FUNCTION_BLOCK FB_StateMachine
VAR_INPUT
    EnableIn : BOOL;
    cfgAutoRun : BOOL;
    inpBlockedCondition : DINT;
    inpStarvedCondition : DINT;
    inpSubmoduleFaulted : BOOL;
END_VAR

VAR_OUTPUT
    EnableOut : BOOL;
    Status : ST_SM_Status;
END_VAR

VAR CONSTANT
    HOMING_MIN   : DINT := 1000; HOMING_MAX   : DINT := 1999;
    RUNNING_MIN  : DINT := 3000; RUNNING_MAX  : DINT := 3999;
    STOPPING_MIN : DINT := 2000; STOPPING_MAX : DINT := 2999;
    ABORTING_MIN : DINT := 5000; ABORTING_MAX : DINT := 5999;
    PAUSING_MIN  : DINT := 4000; PAUSING_MAX  : DINT := 4999;
    PROCEEDING_MIN : DINT := 6000; PROCEEDING_MAX : DINT := 6999;
END_VAR

VAR
    // Internal command request flags (set by methods, consumed by body)
    _abortRequested : BOOL;
    _completeStateRequested : BOOL;
    _homeRequested : BOOL;
    _pauseRequested : BOOL;
    _proceedRequested : BOOL;
    _startRequested : BOOL;
    _stopRequested : BOOL;
    _retryActive : BOOL;
    RetryComplete : BOOL;
    
    // Timer
    StepTimer : TON;
    
    // Edge detection
    R_TRIG_1 : R_TRIG;
    R_TRIG_5 : R_TRIG;
    
    // Internal state tracking
    _previousState : E_SM_State;
    PreviousStep : DINT;
    TimerReset : BOOL;
    LsOdd : DINT;
    _returnState : E_SM_State;
    ReturnNextStep : DINT;
    
    // Permission handlers
    permAuto : FB_Permissives;
    permHome : FB_Permissives;
    permProceed : FB_Permissives;
    permStart : FB_Permissives;
    
    // Running interlock (latching - auto-aborts from any active state)
    intlkRunning : FB_Interlock;
    
    // Temp variables
    permIndex : UDINT;
    stepIsZero : BOOL;
    seqDone : BOOL;
    
    // Source control
    bSourceLockedToProg : BOOL;
    
    // Step ownership (internal)
    _nextStep : DINT;
END_VAR


//-----------------------------------------------------------------------------
// Main Implementation
//-----------------------------------------------------------------------------
EnableOut := EnableIn;

// Only execute if enabled
IF EnableIn THEN
    //-------------------------------------------------------------------------
    // Process permissions for different states
    //-------------------------------------------------------------------------
    permHome();
    permStart();
    permProceed();
    permAuto();
    
    intlkRunning();
    
    // Auto-abort if any running interlock trips (e-stop, safety gate, etc.)
    IF NOT intlkRunning.sts.bOK AND
       NOT (Status.State = E_SM_State.STOPPED OR Status.State = E_SM_State.ABORTING) THEN
        _abortRequested := TRUE;
    END_IF;
    
    //-------------------------------------------------------------------------
    // Ready state calculations
    //-------------------------------------------------------------------------
    Status.ReadyToHome := (Status.State = E_SM_State.STOPPED) AND
                          permHome.sts.bOK AND
                          permAuto.sts.bOK;

    Status.ReadyToStart := (Status.State = E_SM_State.READY) AND
                          permStart.sts.bOK AND
                          permAuto.sts.bOK AND
                          NOT Status.AutoStartRequest;

    Status.ReadyToProceed := (Status.State = E_SM_State.PAUSED) AND
                            permProceed.sts.bOK AND
                            permAuto.sts.bOK;

    //-------------------------------------------------------------------------
    // Auto-start request logic
    // AutoCycle fires when we just finished a RUNNING cycle (READY with LastState=RUNNING)
    //-------------------------------------------------------------------------
    Status.AutoStartRequest := _startRequested AND NOT permStart.sts.bOK;
    Status.AutoCycleRequest := cfgAutoRun AND (Status.State = E_SM_State.READY) AND
                              (Status.LastState = E_SM_State.RUNNING) AND NOT permStart.sts.bOK;

    //-------------------------------------------------------------------------
    // Remember last state before change
    //-------------------------------------------------------------------------
    _previousState := Status.State;

    //-------------------------------------------------------------------------
    // Auto-run handling (internal - not from external command)
    //-------------------------------------------------------------------------
    IF cfgAutoRun AND permAuto.sts.bOK AND permStart.sts.bOK AND
       (Status.State = E_SM_State.READY) AND (Status.LastState = E_SM_State.RUNNING) THEN
        _startRequested := TRUE;
    END_IF;
    
    //-------------------------------------------------------------------------
    // Sequence completion inference
    //-------------------------------------------------------------------------
    seqDone := _IsStepInStateRange(
        state := Status.State,
        nStep := Status.Step.Current
    ) AND (_nextStep = 0);

    R_TRIG_5(CLK := seqDone);
    IF R_TRIG_5.Q THEN
        _completeStateRequested := TRUE;
    END_IF;

    //-------------------------------------------------------------------------
    // State Transitions
    //-------------------------------------------------------------------------

    // Homing complete → Ready
    IF _completeStateRequested AND (Status.State = E_SM_State.HOMING) THEN
        _nextStep := 0;
        Status.State := E_SM_State.READY;
        _completeStateRequested := FALSE;
    END_IF;

    // Running complete → Ready (LastState will be RUNNING so AutoCycle can detect a just-finished cycle)
    IF _completeStateRequested AND (Status.State = E_SM_State.RUNNING) THEN
        _nextStep := 0;
        Status.State := E_SM_State.READY;
        _completeStateRequested := FALSE;
    END_IF;

    // Running + Stop → Stopping
    IF _stopRequested AND (Status.State = E_SM_State.RUNNING) THEN
        Status.State := E_SM_State.STOPPING;
    END_IF;

    // Stopping complete → Stopped
    IF _completeStateRequested AND (Status.State = E_SM_State.STOPPING) THEN
        _nextStep := 0;
        Status.State := E_SM_State.STOPPED;
        _completeStateRequested := FALSE;
    END_IF;

    // Aborting complete → Stopped (Status.Faulted remains indicated via LastState = ABORTING)
    IF _completeStateRequested AND (Status.State = E_SM_State.ABORTING) THEN
        _nextStep := 0;
        Status.State := E_SM_State.STOPPED;
        _completeStateRequested := FALSE;
    END_IF;

    // Running + Pause → Pausing (save context for Proceed)
    IF _pauseRequested AND (Status.State = E_SM_State.RUNNING) THEN
        _returnState := Status.State;
        ReturnNextStep := Status.Step.Current;  // resume re-enters same step
        Status.State := E_SM_State.PAUSING;
        _nextStep := 0;
    END_IF;

    // Pausing complete → Paused
    IF _completeStateRequested AND (Status.State = E_SM_State.PAUSING) THEN
        _nextStep := 0;
        Status.State := E_SM_State.PAUSED;
        _completeStateRequested := FALSE;
    END_IF;

    // Proceeding complete → return to state before pause, re-enter the paused step
    IF _completeStateRequested AND (Status.State = E_SM_State.PROCEEDING) THEN
        _nextStep := ReturnNextStep;
        Status.State := _returnState;
        _completeStateRequested := FALSE;
    END_IF;

    // Ready + Start → Running
    IF (_startRequested OR
        (Status.AutoStartRequest AND permStart.sts.bOK AND permAuto.sts.bOK)) AND
        (Status.State = E_SM_State.READY) THEN
        _nextStep := 0;
        Status.State := E_SM_State.RUNNING;
        _startRequested := FALSE;
    END_IF;

    // Ready + Stop → Stopped (no sequence needed, machine is already quiescent)
    IF _stopRequested AND (Status.State = E_SM_State.READY) THEN
        _nextStep := 0;
        Status.State := E_SM_State.STOPPED;
    END_IF;

    // Stopped + Home → Homing
    IF _homeRequested AND (Status.State = E_SM_State.STOPPED) THEN
        _nextStep := 0;
        Status.State := E_SM_State.HOMING;
    END_IF;

    // Paused + Proceed → Proceeding
    IF _proceedRequested AND (Status.State = E_SM_State.PAUSED) THEN
        _nextStep := 0;
        Status.State := E_SM_State.PROCEEDING;
    END_IF;

    // Abort from any state except Stopped / Aborting
    IF _abortRequested AND NOT (Status.State = E_SM_State.STOPPED OR Status.State = E_SM_State.ABORTING) THEN
        _nextStep := 0;
        Status.State := E_SM_State.ABORTING;
    END_IF;
    
    //-------------------------------------------------------------------------
    // Track state changes
    //-------------------------------------------------------------------------
    IF Status.State <> _previousState THEN
        Status.LastState := _previousState;
    END_IF;
    
    //-------------------------------------------------------------------------
    // Derived status flags
    //-------------------------------------------------------------------------
    Status.WaitingState := (Status.State = E_SM_State.STOPPED) OR (Status.State = E_SM_State.READY) OR
                           (Status.State = E_SM_State.PAUSED);
    Status.ActiveState  := (Status.State = E_SM_State.HOMING) OR (Status.State = E_SM_State.RUNNING) OR
                           (Status.State = E_SM_State.STOPPING) OR (Status.State = E_SM_State.PAUSING) OR
                           (Status.State = E_SM_State.PROCEEDING) OR (Status.State = E_SM_State.ABORTING);

    //-------------------------------------------------------------------------
    // Step and timer management
    //-------------------------------------------------------------------------
    
    // Reset timer and clear step name when transitioning to step 0
    stepIsZero := (Status.Step.Current = 0);
    R_TRIG_1(CLK := stepIsZero);
    IF R_TRIG_1.Q THEN
        Status.Step.Name := '';
        _ClearStepPermissives();
        TimerReset := TRUE;
        StepTimer(IN := FALSE, PT := T#99H);
        Status.Step.TimerSeconds := 0.0;
    END_IF;
    
    // Auto-initialize first step when entering an active state
    IF Status.Step.Current = 0 AND Status.ActiveState THEN
        _nextStep := _GetFirstStepForState(state := Status.State);
    END_IF;
    
    // Detect step change and update
    IF Status.Step.Current <> _nextStep THEN
        PreviousStep := Status.Step.Current;
        Status.Step.Current := _nextStep;
        TimerReset := TRUE;
        StepTimer(IN := FALSE, PT := T#99H);
        Status.Step.TimerSeconds := 0.0;
    END_IF;
    
    Status.Step.Next := _nextStep;
    
    // Step timer logic
    IF NOT (Status.State = E_SM_State.PAUSED) OR ((Status.State = E_SM_State.PAUSED) AND _completeStateRequested) THEN
        IF TimerReset THEN
            StepTimer(IN := FALSE, PT := T#99H);
            Status.Step.TimerSeconds := 0.0;
            TimerReset := FALSE;
        ELSE
            StepTimer(IN := TRUE, PT := T#99H);
            Status.Step.TimerSeconds := UDINT_TO_REAL(TIME_TO_UDINT(StepTimer.ET)) / 1000.0;
        END_IF;
    ELSE
        StepTimer(IN := FALSE, PT := T#99H);
    END_IF;
    
    //-------------------------------------------------------------------------
    // Fault detection
    //-------------------------------------------------------------------------
    LsOdd := Status.Step.Current MOD 2;
    Status.Faulted := LsOdd <> 0;
    Status.SubmoduleFaulted := inpSubmoduleFaulted;
    
    //-------------------------------------------------------------------------
    // Retry logic
    //-------------------------------------------------------------------------
    IF RetryComplete THEN
        _retryActive := FALSE;
        RetryComplete := FALSE;
    END_IF;
    
    IF _retryActive THEN
        RetryComplete := TRUE;
    END_IF;
    
    IF _retryActive AND Status.Faulted THEN
        // Roll back to previous (even, non-faulted) step to re-enter it
        _nextStep := Status.Step.Current - 1;
    END_IF;
    
    //-------------------------------------------------------------------------
    // OEE condition codes (Blocked / Starved)
    //-------------------------------------------------------------------------
    IF inpBlockedCondition = 0 THEN
        Status.BlockedCondition := 0;
    END_IF;
    
    IF inpBlockedCondition <> 0 AND
       (Status.State = E_SM_State.RUNNING OR Status.State = E_SM_State.STOPPING OR
        Status.State = E_SM_State.READY) THEN
        Status.BlockedCondition := inpBlockedCondition;
        inpBlockedCondition := 0;
    END_IF;
    
    IF inpStarvedCondition = 0 THEN
        Status.StarvedCondition := 0;
    END_IF;
    
    IF inpStarvedCondition <> 0 AND
       (Status.State = E_SM_State.RUNNING OR Status.State = E_SM_State.STOPPING OR
        Status.State = E_SM_State.READY) THEN
        Status.StarvedCondition := inpStarvedCondition;
        inpStarvedCondition := 0;
    END_IF;
    
ELSE
    // Reset command requests when disabled
    _startRequested := FALSE;
    _stopRequested := FALSE;
    _homeRequested := FALSE;
    _abortRequested := FALSE;
    _pauseRequested := FALSE;
    _proceedRequested := FALSE;
    _completeStateRequested := FALSE;
    Status.Step.Name := '';
        _ClearStepPermissives();
END_IF;

METHOD PRIVATE _ClearStepPermissives
Status.Step.PermCfg.nBypassable := 0;
Status.Step.PermStatus.bOK := FALSE;
Status.Step.PermStatus.nPermissives := 0;
Status.Step.PermStatus.nBypassMask := 0;
Status.Step.PermStatus.nFirstFailureBitIndex := 999;

FOR permIndex := 0 TO 63 DO
        Status.Step.PermCfg.aNames[permIndex] := '';
        Status.Step.PermStatus.aFaceplates[permIndex].name := '';
        Status.Step.PermStatus.aFaceplates[permIndex].stsOK := FALSE;
        Status.Step.PermStatus.aFaceplates[permIndex].stsMapped := FALSE;
        Status.Step.PermStatus.aFaceplates[permIndex].stsBypassed := FALSE;
        Status.Step.PermStatus.aFaceplates[permIndex].cfgBypassable := FALSE;
END_FOR;
END_METHOD

METHOD PRIVATE _GetFirstStepForState : DINT
VAR_INPUT
        state : E_SM_State;
END_VAR
CASE state OF
        E_SM_State.HOMING:     _GetFirstStepForState := HOMING_MIN;
        E_SM_State.RUNNING:    _GetFirstStepForState := RUNNING_MIN;
        E_SM_State.STOPPING:   _GetFirstStepForState := STOPPING_MIN;
        E_SM_State.ABORTING:   _GetFirstStepForState := ABORTING_MIN;
        E_SM_State.PAUSING:    _GetFirstStepForState := PAUSING_MIN;
        E_SM_State.PROCEEDING: _GetFirstStepForState := PROCEEDING_MIN;
ELSE
        _GetFirstStepForState := 0;
END_CASE;
END_METHOD

METHOD PRIVATE _GetLastStepForState : DINT
VAR_INPUT
        state : E_SM_State;
END_VAR
CASE state OF
        E_SM_State.HOMING:     _GetLastStepForState := HOMING_MAX;
        E_SM_State.RUNNING:    _GetLastStepForState := RUNNING_MAX;
        E_SM_State.STOPPING:   _GetLastStepForState := STOPPING_MAX;
        E_SM_State.ABORTING:   _GetLastStepForState := ABORTING_MAX;
        E_SM_State.PAUSING:    _GetLastStepForState := PAUSING_MAX;
        E_SM_State.PROCEEDING: _GetLastStepForState := PROCEEDING_MAX;
ELSE
        _GetLastStepForState := 0;
END_CASE;
END_METHOD

METHOD PRIVATE _IsStepInStateRange : BOOL
VAR_INPUT
        state : E_SM_State;
        nStep : DINT;
END_VAR
_IsStepInStateRange := (nStep >= _GetFirstStepForState(state := state)) AND
                                             (nStep <= _GetLastStepForState(state := state));
END_METHOD

{attribute 'TcRpcEnable' := '1'}
METHOD Abort : E_RpcMethodResponse
VAR_INPUT
    eRequester : E_Requester := E_Requester.PROG;
END_VAR
// Safety command - skip source check, skip fault check
IF Status.State = E_SM_State.STOPPED OR Status.State = E_SM_State.ABORTING THEN
    Abort := E_RpcMethodResponse.REJECTED_WRONG_STATE;
    RETURN;
END_IF;

// Execute - clear other requests, set abort
_startRequested := FALSE;
_stopRequested := FALSE;
_homeRequested := FALSE;
_pauseRequested := FALSE;
_proceedRequested := FALSE;
_completeStateRequested := FALSE;
_abortRequested := TRUE;
Abort := E_RpcMethodResponse.ACCEPTED;
END_METHOD

{attribute 'TcRpcEnable' := '1'}
METHOD Home : E_RpcMethodResponse
VAR_INPUT
    eRequester : E_Requester := E_Requester.PROG;
END_VAR
// Common validation
Home := F_ValidateRequester(eRequester, bSourceLockedToProg, Status.Faulted, FALSE, FALSE);
IF Home <> E_RpcMethodResponse.ACCEPTED THEN RETURN; END_IF;

// State check
IF NOT (Status.State = E_SM_State.STOPPED) THEN
    Home := E_RpcMethodResponse.REJECTED_WRONG_STATE;
    RETURN;
END_IF;

// Permission check (Home-specific)
IF NOT permHome.sts.bOK THEN
    Home := E_RpcMethodResponse.REJECTED_PERMISSIVE_NOT_MET;
    RETURN;
END_IF;

// Permission check (global auto permissives)
IF NOT permAuto.sts.bOK THEN
    Home := E_RpcMethodResponse.REJECTED_PERMISSIVE_NOT_MET;
    RETURN;
END_IF;

// Execute
_abortRequested := FALSE;
_pauseRequested := FALSE;
_proceedRequested := FALSE;
_startRequested := FALSE;
_stopRequested := FALSE;
_completeStateRequested := FALSE;
_homeRequested := TRUE;
Home := E_RpcMethodResponse.ACCEPTED;
END_METHOD

METHOD LockSource
VAR_INPUT
    bLock : BOOL;
END_VAR
bSourceLockedToProg := bLock;
END_METHOD

{attribute 'TcRpcEnable' := '1'}
METHOD Pause : E_RpcMethodResponse
VAR_INPUT
    eRequester : E_Requester := E_Requester.PROG;
END_VAR
// Common validation
Pause := F_ValidateRequester(eRequester, bSourceLockedToProg, Status.Faulted, FALSE, FALSE);
IF Pause <> E_RpcMethodResponse.ACCEPTED THEN RETURN; END_IF;

// State check
IF NOT (Status.State = E_SM_State.RUNNING) THEN
    Pause := E_RpcMethodResponse.REJECTED_WRONG_STATE;
    RETURN;
END_IF;

// Execute
_abortRequested := FALSE;
_homeRequested := FALSE;
_proceedRequested := FALSE;
_startRequested := FALSE;
_stopRequested := FALSE;
_completeStateRequested := FALSE;
_pauseRequested := TRUE;
Pause := E_RpcMethodResponse.ACCEPTED;
END_METHOD

{attribute 'TcRpcEnable' := '1'}
METHOD Proceed : E_RpcMethodResponse
VAR_INPUT
    eRequester : E_Requester := E_Requester.PROG;
END_VAR
// Common validation
Proceed := F_ValidateRequester(eRequester, bSourceLockedToProg, Status.Faulted, FALSE, FALSE);
IF Proceed <> E_RpcMethodResponse.ACCEPTED THEN RETURN; END_IF;

// State check
IF NOT (Status.State = E_SM_State.PAUSED) THEN
    Proceed := E_RpcMethodResponse.REJECTED_WRONG_STATE;
    RETURN;
END_IF;

// Permission check (Proceed-specific)
IF NOT permProceed.sts.bOK THEN
    Proceed := E_RpcMethodResponse.REJECTED_PERMISSIVE_NOT_MET;
    RETURN;
END_IF;

// Permission check (global auto permissives)
IF NOT permAuto.sts.bOK THEN
    Proceed := E_RpcMethodResponse.REJECTED_PERMISSIVE_NOT_MET;
    RETURN;
END_IF;

// Execute
_abortRequested := FALSE;
_homeRequested := FALSE;
_pauseRequested := FALSE;
_startRequested := FALSE;
_stopRequested := FALSE;
_completeStateRequested := FALSE;
_proceedRequested := TRUE;
Proceed := E_RpcMethodResponse.ACCEPTED;
END_METHOD

{attribute 'TcRpcEnable' := '1'}
METHOD Retry : E_RpcMethodResponse
VAR_INPUT
    eRequester : E_Requester := E_Requester.PROG;
END_VAR
// Common validation
Retry := F_ValidateRequester(eRequester, bSourceLockedToProg, Status.Faulted, FALSE, FALSE);
IF Retry <> E_RpcMethodResponse.ACCEPTED THEN RETURN; END_IF;

// Execute - set retry directly
_retryActive := TRUE;
Retry := E_RpcMethodResponse.ACCEPTED;
END_METHOD

{attribute 'TcRpcEnable' := '1'}
METHOD Start : E_RpcMethodResponse
VAR_INPUT
    eRequester : E_Requester := E_Requester.PROG;
END_VAR
// Common validation
Start := F_ValidateRequester(eRequester, bSourceLockedToProg, Status.Faulted, FALSE, FALSE);
IF Start <> E_RpcMethodResponse.ACCEPTED THEN RETURN; END_IF;

// State check
IF NOT (Status.State = E_SM_State.READY) THEN
    Start := E_RpcMethodResponse.REJECTED_WRONG_STATE;
    RETURN;
END_IF;

// Permission check (Start-specific)
IF NOT permStart.sts.bOK THEN
    Start := E_RpcMethodResponse.REJECTED_PERMISSIVE_NOT_MET;
    RETURN;
END_IF;

// Permission check (global auto permissives)
IF NOT permAuto.sts.bOK THEN
    Start := E_RpcMethodResponse.REJECTED_PERMISSIVE_NOT_MET;
    RETURN;
END_IF;

// Execute
_abortRequested := FALSE;
_pauseRequested := FALSE;
_homeRequested := FALSE;
_proceedRequested := FALSE;
_stopRequested := FALSE;
_completeStateRequested := FALSE;
_startRequested := TRUE;
Start := E_RpcMethodResponse.ACCEPTED;
END_METHOD

{attribute 'TcRpcEnable' := '1'}
METHOD Stop : E_RpcMethodResponse
VAR_INPUT
    eRequester : E_Requester := E_Requester.PROG;
END_VAR
// Safety command - skip source check, skip fault check
IF Status.State = E_SM_State.STOPPED OR Status.State = E_SM_State.STOPPING THEN
    Stop := E_RpcMethodResponse.REJECTED_WRONG_STATE;
    RETURN;
END_IF;

// Execute
_abortRequested := FALSE;
_homeRequested := FALSE;
_proceedRequested := FALSE;
_startRequested := FALSE;
_pauseRequested := FALSE;
_completeStateRequested := FALSE;
_stopRequested := TRUE;
Stop := E_RpcMethodResponse.ACCEPTED;
END_METHOD

{attribute 'TcRpcEnable' := '1'}
// Map a running interlock bit. Call every cycle. bGood=TRUE means the condition is safe.
// If bGood goes FALSE from any non-stopped state the machine auto-aborts.
METHOD MapRunningIntlk
VAR_INPUT
    bitIndex : UDINT;
    bGood    : BOOL;
END_VAR
intlkRunning.MapInput(bitIndex := bitIndex, inputValue := bGood);
END_METHOD

{attribute 'TcRpcEnable' := '1'}
// Clear latched running interlock bits after the real-world condition has recovered.
// The machine will still be in STOPPED/ABORTING — issue Home/Start separately.
METHOD ResetRunningIntlk
intlkRunning.Reset();
END_METHOD

// INTERNAL: used by FB_Step to advance the sequence. Not part of the user API.
METHOD INTERNAL SetNextStep
VAR_INPUT
    nStep : DINT;
END_VAR
_nextStep := nStep;
END_METHOD

// INTERNAL: used by FB_Step to publish its name to StepInfo. Not part of the user API.
METHOD INTERNAL SetStepName
VAR_INPUT
    sName : STRING(40);
END_VAR
Status.Step.Name := sName;
END_METHOD

// INTERNAL: used by FB_Step to publish the active step permissive data for HMI / OPC.
METHOD INTERNAL SetStepPermissives
VAR_INPUT
        cfg : ST_Permissive_Config;
        sts : ST_Permissive_Status;
END_VAR
Status.Step.PermCfg := cfg;
Status.Step.PermStatus := sts;
END_METHOD

// INTERNAL: used by FB_Step to fault the current step (timeout, etc.).
// Faults by advancing to the next (odd) step number -- Status.Faulted derives
// from (CurrentStep MOD 2). Not part of the user API.
METHOD INTERNAL SetStepFault
VAR_INPUT
    bFault : BOOL;
END_VAR
IF bFault THEN
    _nextStep := Status.Step.Current + 1;
END_IF;
END_METHOD

END_FUNCTION_BLOCK

(* stored: Version 1.1.0.1, ProductVersion 3.1.4026.12
   POU FB_StateMachine: Id {7408693c-f749-4b9e-8684-bfcba9889df8}, SpecialFunc None
   Folder Public: Id {f0c10001-0001-0001-0001-000000000001}
   Folder Internal: Id {f0c10002-0001-0001-0001-000000000002}
   Folder Private: Id {f0c10003-0001-0001-0001-000000000003}
   Method _ClearStepPermissives: Id {d4e5f6a7-b8c9-0123-def0-123456789abf}
   Method _GetFirstStepForState: Id {d4e5f6a7-b8c9-0123-def0-123456789ac0}
   Method _GetLastStepForState: Id {d4e5f6a7-b8c9-0123-def0-123456789ac1}
   Method _IsStepInStateRange: Id {d4e5f6a7-b8c9-0123-def0-123456789ac2}
   Method Abort: Id {c1234567-1234-1234-1234-12345678C001}
   Method Home: Id {c1234567-1234-1234-1234-12345678C002}
   Method LockSource: Id {c1234567-1234-1234-1234-12345678C008}
   Method Pause: Id {c1234567-1234-1234-1234-12345678C003}
   Method Proceed: Id {c1234567-1234-1234-1234-12345678C004}
   Method Retry: Id {c1234567-1234-1234-1234-12345678C005}
   Method Start: Id {c1234567-1234-1234-1234-12345678C006}
   Method Stop: Id {c1234567-1234-1234-1234-12345678C007}
   Method MapRunningIntlk: Id {f7a8b9c0-d1e2-4f30-a001-000000000001}
   Method ResetRunningIntlk: Id {f7a8b9c0-d1e2-4f30-a001-000000000002}
   Method SetNextStep: Id {d4e5f6a7-b8c9-0123-def0-123456789abc}
   Method SetStepName: Id {d4e5f6a7-b8c9-0123-def0-123456789abd}
   Method SetStepPermissives: Id {d4e5f6a7-b8c9-0123-def0-123456789abe}
   Method SetStepFault: Id {e5f6a7b8-c9d0-1234-ef01-23456789abcd} *)
